{attribute 'qualified_only'}
VAR_GLOBAL
	In AT %I*:WeldRobotIn;
	Out AT %Q*:WeldRobotOut;
END_VAR

(* stored: Version 1.1.0.1, ProductVersion 3.1.4024.16
   GVL WeldRobot: Id {1d5b7808-61b8-48d7-80f6-17cad38f58c0} *)
